GLOBALCONSTANTS Override_K (* K-Werte fuer AX_AUI_MUX_3 in Override_K_Select (0=Normal, 1=Force FALSE, 2=Force TRUE) *)
  (* Standard: 61499-1; Description: Copyright (c) 2026 HR Agrartechnik GmbH This program and the accompanying materials are made available under the terms of the Eclipse Public License 2.0 which is available at https://www.eclipse.org/legal/epl-2.0/ SPDX-License-Identifier: EPL-2.0 *)
  (* Version 1.0, 2026-08-13, Franz Höpfinger, HR Agrartechnik GmbH *)
  PACKAGE adapter::OverrideK::const;
  VAR_GLOBAL CONSTANT
    Override_K_Normal : UINT := UINT#0; (* K=0, AX_AUI_MUX_3.IN1 (Normal/Eingang) *)
    Override_K_ForceFalse : UINT := UINT#1; (* K=1, AX_AUI_MUX_3.IN2 (Force FALSE / Voll) *)
    Override_K_ForceTrue : UINT := UINT#2; (* K=2, AX_AUI_MUX_3.IN3 (Force TRUE / Leer) *)
  END_VAR
END_GLOBALCONSTANTS
